// TIA Portal V20 export
TYPE "LConSMC_typeFrictionMeasurementV2Out"
// stored: Access Published
   STRUCT
      done { ExternalWritable := 'False'} : Bool;   // TRUE: Die Messung wurde erfolgreich beendet / TRUE: Measurement is finished
      valid : Bool;   // TRUE: Die Messwerte sind gültig / TRUE: Measurement values are valid
      aborted : Bool;   // TRUE: Die Messung wurde abgebrochen / TRUE: Measuremetn was aborted
      busy { ExternalWritable := 'False'} : Bool;   // TRUE: Die Messung ist aktiv / TRUE: Measurement is active
      error { ExternalWritable := 'False'} : Bool;   // TRUE: Es ist ein Fehler aufgetreten / TRUE: An error has occured
      subfunctionState : Word;   // Detaillierte Fehlerbeschreibung / Error identification
      status { ExternalWritable := 'False'} : Word := 16#7000;   // Aktueller Status des Funktionsbausteins / Current status of function block
   END_STRUCT;
END_TYPE
